# EPICS substitutions: tgpApp/Db/tpg36x.substitutions
file "tpgx6x.template" {
  pattern
    {P,    DEVICE, "IFPRESSUR1", "IFPRESSUR2", "PORT", "RECSIM", "DISABLE"}

    {"\$(P)", "TPG36x", "\$(IFPRESSUR1)", "\$(IFPRESSUR2)", "\$(PORT)", "\$(RECSIM)", "\$(DISABLE)"}
}
